{attribute 'GeneratedUsingTerminal: EK1960-0000-0019'}
{attribute addProperty BoxType "EK1960-0000-0019"}
{attribute addProperty Id "EMPTY_STRUCTURE"}
{attribute addProperty CRC "0"}
{attribute addProperty Size "0"}
TYPE EMPTY_STRUCTURE :
STRUCT
END_STRUCT
END_TYPE

(* stored: Version 1.2.0.0, ProductVersion 3.1.4024.9
   DUT EMPTY_STRUCTURE: Id {8654bd2d-bbdc-421f-aa68-62023bf9b040} *)
